PROGRAM ST00_ChangeRecipe
VAR
	iStep : INT;
END_VAR

END_PROGRAM

(* stored: Version 1.1.0.1, ProductVersion 3.1.4024.11
   POU ST00_ChangeRecipe: Id {fb9028b9-dede-4a2a-8dbe-fcfb9953b31e}, SpecialFunc None *)
